Fanuc KAREL source: ko00026.KL

-- PROVISIONAL review KL for V770-1; original PC SHA256 dcfce9d0b95b098562ed074ccd55163826f070d52c860504ad1c195dd26f79b4
-- Incomplete behavior may be omitted. Consult companion uncertainty JSON. Do not deploy.
PROGRAM KO00026
%NOLOCKGROUP
-- UNRESOLVED_DECL P1 type=000199
-- UNRESOLVED_DECL P2 type=000199
-- UNRESOLVED_DECL P3 type=000199
-- UNRESOLVED_DECL OUT type=000102
BEGIN
  -- UNRESOLVED_PC offsets 5-65; opcodes 27,27,49,7E,AD,27,49,7E,AD,27,49,7E,AD,76,7E,4A
  -- UNRESOLVED_PC offsets 70-74; opcodes 7F
END KO00026
